FUNCTION Convert_LWORD_TO_LINT : Hresult
VAR_INPUT
	in : LWORD;
	out : REFERENCE TO LINT;
END_VAR
VAR
	converted : LINT;
END_VAR
VAR CONSTANT
	INCOMPATIBLE : HRESULT := 16#9811070E;
END_VAR

converted := LWORD_TO_LINT(in);

IF (LINT_TO_LWORD(converted) <> in) THEN
	Convert_LWORD_TO_LINT := INCOMPATIBLE;
	RETURN;
END_IF

out := converted;

END_FUNCTION

(* stored: Version 1.1.0.1, ProductVersion 3.1.4024.12
   POU Convert_LWORD_TO_LINT: Id {29f039ec-2e19-4450-aee3-9a4ef4cc0a25}, SpecialFunc None *)
